// SIMATIC S7-200 SMART project (STEP 7-Micro/WIN SMART), CPU ST20

SYMBOL_TABLE System Symbols
Always_On        SM0.0    // Always ON
END_SYMBOL_TABLE

ORGANIZATION_BLOCK MAIN:OB1
TITLE=Program Comments
BEGIN
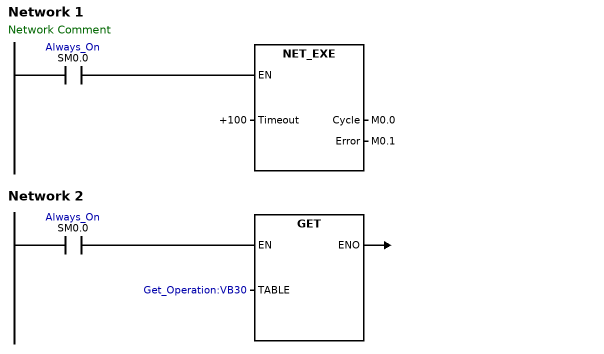
Network 1
// Network Comment
LD     Always_On:SM0.0
CALL   NET_EXE:SBR1, +100, M0.0, M0.1
Network 2
LD     Always_On:SM0.0
GET    Get_Operation:VB30
END_ORGANIZATION_BLOCK

// SBR1: protected block, not included
